{attribute addProperty BoxType "EL6080-0000-0016"}
{attribute addProperty Id "ControlAT %Q*ARRAY [0..1] OF USINT00"}
{attribute addProperty CRC "2871997638"}
{attribute addProperty SizeInBites "0"}
{attribute addProperty SizeInBytes "0"}
TYPE Control_AB2F34C6 :
STRUCT
	{attribute addProperty Name "Control"}
	Control AT %Q* : ARRAY [0..1] OF USINT;
END_STRUCT
END_TYPE

(* stored: Version 1.2.0.0, ProductVersion 3.1.4024.9
   DUT Control_AB2F34C6: Id {749ab2f3-a42f-457f-b305-f67ae26b530d} *)
